(* Logix 5000 project; controller DCMGSG vendor 1 type 14 code 94 rev 20.12; software revision 20.01 *)
// Handles Scenario Generation I/O for DCMG.

TASK MainTask (continuous, watchdog 500 ms) : MainProgram

MODULES
   Local : vendor 1 type 14 code 94 (ICP 0, rev 20.12)
      SG_OB32_1 : 1756-OB32 (ICP 8, rev 3.3, Output RPI 20 ms)   // Digital output for DCMG Scenario Generator
      SG_OB32_2 : 1756-OB32 (ICP 9, rev 3.3, Output RPI 20 ms)   // Digital output for DCMG Scenario Generator. Signals 33 and up.
      EnvironmentSignals : 1756-OF4 (ICP 7, rev 1.1, Output RPI 12 ms)   // Signals for solar lamp dimming and turbine motor control.
      ETHERNET : 1756-EN2T (ICP 1, Ethernet 192.168.56.222, rev 3.1)
END_MODULES

VAR_GLOBAL   (* controller tags *)
   BRANCH_1_BUS_1_DISTAL_NC : ALIAS FOR Local:8:O.Data.22;
   BRANCH_1_BUS_1_DISTAL_NO : ALIAS FOR Local:8:O.Data.21;
   BRANCH_1_BUS_1_FAULT : ALIAS FOR Local:8:O.Data.23;
   BRANCH_1_BUS_1_LOAD_1_NC : ALIAS FOR Local:8:O.Data.7;
   BRANCH_1_BUS_1_LOAD_1_NO : ALIAS FOR Local:8:O.Data.6;
   BRANCH_1_BUS_1_LOAD_2_NC : ALIAS FOR Local:8:O.Data.5;
   BRANCH_1_BUS_1_LOAD_2_NO : ALIAS FOR Local:8:O.Data.4;
   BRANCH_1_BUS_1_LOAD_3_NC : ALIAS FOR Local:8:O.Data.0;
   BRANCH_1_BUS_1_LOAD_3_NO : ALIAS FOR Local:8:O.Data.3;
   BRANCH_1_BUS_1_PROXIMAL_NC : ALIAS FOR Local:8:O.Data.2;
   BRANCH_1_BUS_1_PROXIMAL_NO : ALIAS FOR Local:8:O.Data.1;
   BRANCH_1_BUS_2_DISTAL_NC : ALIAS FOR Local:9:O.Data.4;
   BRANCH_1_BUS_2_DISTAL_NO : ALIAS FOR Local:9:O.Data.5;
   BRANCH_1_BUS_2_FAULT : ALIAS FOR Local:9:O.Data.8;
   BRANCH_1_BUS_2_LOAD_1_NC : ALIAS FOR Local:8:O.Data.31;
   BRANCH_1_BUS_2_LOAD_1_NO : ALIAS FOR Local:9:O.Data.0;
   BRANCH_1_BUS_2_LOAD_2_NC : ALIAS FOR Local:9:O.Data.1;
   BRANCH_1_BUS_2_LOAD_2_NO : ALIAS FOR Local:9:O.Data.2;
   BRANCH_1_BUS_2_LOAD_3_NC : ALIAS FOR Local:9:O.Data.6;
   BRANCH_1_BUS_2_LOAD_3_NO : ALIAS FOR Local:9:O.Data.7;
   BRANCH_1_BUS_2_PROXIMAL_NC : ALIAS FOR Local:8:O.Data.25;
   BRANCH_1_BUS_2_PROXIMAL_NO : ALIAS FOR Local:8:O.Data.26;
   BRANCH_1_INTERCONNECT_1_FAULT : ALIAS FOR Local:8:O.Data.24;
   BRANCH_1_INTERCONNECT_2_FAULT : ALIAS FOR Local:9:O.Data.9;
   BRANCH_2_BUS_1_DISTAL_NC : ALIAS FOR Local:8:O.Data.9;
   BRANCH_2_BUS_1_DISTAL_NO : ALIAS FOR Local:8:O.Data.10;
   BRANCH_2_BUS_1_FAULT : ALIAS FOR Local:8:O.Data.29;
   BRANCH_2_BUS_1_LOAD_1_NC : ALIAS FOR Local:8:O.Data.15;
   BRANCH_2_BUS_1_LOAD_1_NO : ALIAS FOR Local:8:O.Data.8;
   BRANCH_2_BUS_1_LOAD_2_NC : ALIAS FOR Local:8:O.Data.16;
   BRANCH_2_BUS_1_LOAD_2_NO : ALIAS FOR Local:8:O.Data.14;
   BRANCH_2_BUS_1_LOAD_3_NC : ALIAS FOR Local:8:O.Data.18;
   BRANCH_2_BUS_1_LOAD_3_NO : ALIAS FOR Local:8:O.Data.17;
   BRANCH_2_BUS_1_PROXIMAL_NC : ALIAS FOR Local:8:O.Data.11;
   BRANCH_2_BUS_1_PROXIMAL_NO : ALIAS FOR Local:8:O.Data.12;
   BRANCH_2_BUS_2_DISTAL_NC : ALIAS FOR Local:9:O.Data.13;
   BRANCH_2_BUS_2_DISTAL_NO : ALIAS FOR Local:9:O.Data.14;
   BRANCH_2_BUS_2_FAULT : ALIAS FOR Local:9:O.Data.11;
   BRANCH_2_BUS_2_LOAD_1_NC : ALIAS FOR Local:9:O.Data.20;
   BRANCH_2_BUS_2_LOAD_1_NO : ALIAS FOR Local:9:O.Data.12;
   BRANCH_2_BUS_2_LOAD_2_NC : ALIAS FOR Local:9:O.Data.18;
   BRANCH_2_BUS_2_LOAD_2_NO : ALIAS FOR Local:9:O.Data.19;
   BRANCH_2_BUS_2_LOAD_3_NC : ALIAS FOR Local:9:O.Data.16;
   BRANCH_2_BUS_2_LOAD_3_NO : ALIAS FOR Local:9:O.Data.17;
   BRANCH_2_BUS_2_PROXIMAL_NC : ALIAS FOR Local:8:O.Data.28;
   BRANCH_2_BUS_2_PROXIMAL_NO : ALIAS FOR Local:8:O.Data.27;
   BRANCH_2_INTERCONNECT_1_FAULT : ALIAS FOR Local:8:O.Data.30;
   BRANCH_2_INTERCONNECT_2_FAULT : ALIAS FOR Local:9:O.Data.10;
   CROSSTIE_1_NC : ALIAS FOR Local:8:O.Data.20;
   CROSSTIE_1_NO : ALIAS FOR Local:8:O.Data.19;
   CROSSTIE_2_NC : ALIAS FOR Local:9:O.Data.3;
   CROSSTIE_2_NO : ALIAS FOR Local:9:O.Data.15;
   MAIN_BUS_FAULT : ALIAS FOR Local:8:O.Data.13;
   SolarSetpoint1Alias : ALIAS FOR Local:7:O.Ch0Data;
   SOURCE_1_NC : ALIAS FOR Local:9:O.Data.21;
   SOURCE_2_NC : ALIAS FOR Local:9:O.Data.22;
   SOURCE_3_NC : ALIAS FOR Local:9:O.Data.23;
   SOURCE_4_NC : ALIAS FOR Local:9:O.Data.24;
   SOURCE_5_NC : ALIAS FOR Local:9:O.Data.25;
   SOURCE_6_NC : ALIAS FOR Local:9:O.Data.26;
END_VAR

PROGRAM MainProgram   (* main routine MainRoutine *)

ROUTINE ENVIRONMENT   (* ladder *)
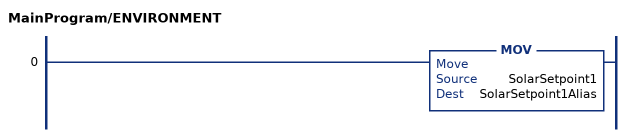
   0: MOV(SolarSetpoint1,SolarSetpoint1Alias);
END_ROUTINE

ROUTINE MainRoutine   (* ladder *)
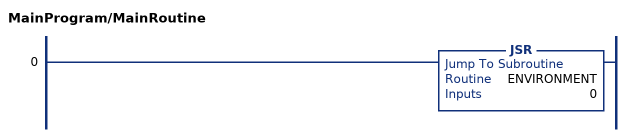
   0: JSR(ENVIRONMENT,0);
END_ROUTINE
END_PROGRAM
